(* PLC project mtcs_safety, Institute of Astronomy Onto 0.0.1 *)
(* stored: creationDateTime 2024-10-22T16:57:18.797943, modificationDateTime 2024-10-22T16:57:18.797943 *)

TYPE SafetyParts : STRUCT
  hydraulics : SafetyHydraulics;  (* Hydraulics safety *)
  emergencyStops : SafetyEmergencyStops;  (* Emergency stops *)
  domeAccess : SafetyDomeAccess;  (* Dome access *)
  motionBlocking : SafetyMotionBlocking;  (* Motion blocking *)
  domeShutter : SafetyDomeShutter;  (* Dome Shutter *)
  io : SafetyIO;  (* I/O modules *)
  configManager : ConfigManager;  (* The config manager (to load/save/activate configuration data) *)
END_STRUCT;
END_TYPE

TYPE SafetyIOParts : STRUCT
  domeAccess : SafetyDomeAccessIO;  (* DA: Dome access I/O *)
  hydraulicsAndSafety : SafetyHydraulicsAndSafetyIO;  (* HS: Hydraulics and Safety I/O *)
END_STRUCT;
END_TYPE

TYPE SafetyHydraulicsAndSafetyIOParts : STRUCT
  COU : EtherCatDevice;  (* HS:COU (EK1101) *)
  DO1 : EtherCatDevice;  (* HS:DO1 (EL2008) *)
  SI1 : EtherCatDevice;  (* HS:SI1 (EL1904) *)
  SI2 : EtherCatDevice;  (* HS:SI2 (EL1904) *)
  SI3 : EtherCatDevice;  (* HS:SI3 (EL1904) *)
  SI4 : EtherCatDevice;  (* HS:SI4 (EL1904) *)
  SL : EtherCatDevice;  (* HS:SL (EL6900) *)
  SO1 : EtherCatDevice;  (* HS:SO1 (EL2904) *)
  AI1 : EtherCatDevice;  (* HS:AI1 (EL3102) *)
  AI2 : EtherCatDevice;  (* HS:AI2 (EL3152) *)
  RTD1 : EtherCatDevice;  (* HS:RTD1 (EL3202-0010) *)
  PWR1 : EtherCatDevice;  (* HS:PWR1 (EL9410) *)
  AO1 : EtherCatDevice;  (* HS:AO1 (EL4132) *)
END_STRUCT;
END_TYPE

TYPE SafetyDomeAccessIOParts : STRUCT
  COU : EtherCatDevice;  (* DA:COU (EK1101) *)
  DI1 : EtherCatDevice;  (* DA:DI1 (EL1008) *)
  DI2 : EtherCatDevice;  (* DA:DI2 (EL1008) *)
  DO1 : EtherCatDevice;  (* DA:DO1 (EL2008) *)
  SI1 : EtherCatDevice;  (* DA:SI1 (EL1904) *)
  RE1 : EtherCatDevice;  (* DA:RE1 (EL2622) *)
  RE2 : EtherCatDevice;  (* DA:RE2 (EL2622) *)
END_STRUCT;
END_TYPE

TYPE SafetyDomeAccessParts : STRUCT
  lampsRelay1 : SimpleRelay;  (* Lamps relay 1 *)
  lampsRelay2 : SimpleRelay;  (* Lamps relay 2 *)
  lampsRelay3 : SimpleRelay;  (* Lamps relay 3 *)
  lampsRelay4 : SimpleRelay;  (* Lamps relay 4 *)
END_STRUCT;
END_TYPE

TYPE SafetyProcesses : STRUCT
  initialize : Process;  (* Start initializing *)
  lock : Process;  (* Lock the system *)
  unlock : Process;  (* Unlock the system *)
  changeOperatingState : ChangeOperatingStateProcess;  (* Change the operating state (e.g. AUTO, MANUAL, ...) *)
END_STRUCT;
END_TYPE

TYPE SafetyHydraulicsProcesses : STRUCT
  startupPumps : Process;  (* Start up the pumps (this will first trigger a reset() command!) *)
  reset : Process;  (* Reset the errors (including the programmed ones and the TwinSAFE group ones) *)
END_STRUCT;
END_TYPE

TYPE SafetyEmergencyStopsProcesses : STRUCT
  reset : Process;  (* Reset the errors (including the programmed ones and the TwinSAFE group ones) *)
END_STRUCT;
END_TYPE

TYPE SafetyDomeAccessProcesses : STRUCT
  reset : Process;  (* Reset the errors (including the programmed ones and the TwinSAFE group ones) *)
  personHasLeft : Process;  (* Unblock the telescope (if possible, i.e. if no E-Stops are active etc.) *)
  bypass : Process;  (* Bypass the doors sensors for the number of seconds defined in the config *)
  bypassPermanently : Process;  (* Bypass the doors sensors permanently (until re-initialization) *)
  stopBypassing : Process;  (* Stop bypassing the doors sensors *)
END_STRUCT;
END_TYPE

TYPE SafetyMotionBlockingProcesses : STRUCT
  reset : Process;  (* Reset the errors (including the programmed ones and the TwinSAFE group ones) *)
END_STRUCT;
END_TYPE

TYPE SafetyDomeShutterProcesses : STRUCT
  reset : Process;  (* Reset the errors (including the programmed ones and the TwinSAFE group ones) *)
END_STRUCT;
END_TYPE

TYPE SafetyStatuses : STRUCT
  initializationStatus : InitializationStatus;
  healthStatus : HealthStatus;
  busyStatus : BusyStatus;
  operatingStatus : OperatingStatus;
  communicationHealthStatus : HealthStatus;
  functionBlockHealthStatus : HealthStatus;
  outputHealthStatus : HealthStatus;
END_STRUCT;
END_TYPE

TYPE SafetyIOStatuses : STRUCT
  healthStatus : HealthStatus;  (* Is the I/O in a healthy state? *)
END_STRUCT;
END_TYPE

TYPE SafetyHydraulicsAndSafetyIOStatuses : STRUCT
  healthStatus : HealthStatus;  (* Is the I/O in a healthy state? *)
END_STRUCT;
END_TYPE

TYPE SafetyDomeAccessIOStatuses : STRUCT
  healthStatus : HealthStatus;  (* Is the I/O in a healthy state? *)
END_STRUCT;
END_TYPE

TYPE SafetyHydraulicsStatuses : STRUCT
  healthStatus : HealthStatus;  (* Is the safety in a healthy state? Good=RUN, Bad=safe stopped *)
  busyStatus : BusyStatus;  (* Is the safety busy? *)
END_STRUCT;
END_TYPE

TYPE SafetyEmergencyStopsStatuses : STRUCT
  healthStatus : HealthStatus;  (* Are the emergency stops in a healthy state? Good=RUN, Bad=safe stopped *)
  busyStatus : BusyStatus;  (* Is the safety busy? *)
END_STRUCT;
END_TYPE

TYPE SafetyDomeAccessStatuses : STRUCT
  healthStatus : HealthStatus;  (* Are the emergency stops in a healthy state? Good=RUN, Bad=safe stopped *)
  busyStatus : BusyStatus;  (* Is the safety busy? *)
END_STRUCT;
END_TYPE

TYPE SafetyMotionBlockingStatuses : STRUCT
  busyStatus : BusyStatus;  (* Is the safety busy? *)
  healthStatus : HealthStatus;  (* Is everything unblocked? Good=unblocked, Bad=safe stopped *)
END_STRUCT;
END_TYPE

TYPE SafetyDomeShutterStatuses : STRUCT
  busyStatus : BusyStatus;  (* Is the safety busy? *)
  healthStatus : HealthStatus;  (* Is everything unblocked? Good=unblocked, Bad=safe stopped *)
END_STRUCT;
END_TYPE

TYPE SafetyDomeAccessAlertConfig : STRUCT
  pattern : UDINT;  (* Bit pattern, for which bit=high means alert active, bit=low means alert off *)
  patternLength : USINT;  (* Number of bits of the bitPattern to use (between 1 and 32) *)
  bitLength : UINT;  (* Sound length of 1 bit, in milliseconds *)
  totalTime : UINT;  (* The time, in number of milliseconds, during which the pattern is repeated. 0 means repeat forever. *)
END_STRUCT;
END_TYPE

TYPE SafetyDomeAccessConfig : STRUCT
  disabled : BOOL;  (* True if the dome access control system should be disabled permanently. *)
  bypassTimeAfterPassword : LREAL;  (* Time until during which the doors sensors are being bypassed after entering the password, in seconds *)
  bypassingSound : SafetyDomeAccessAlertConfig;  (* Sound to play when the doors sensors are being bypassed *)
  bypassedPermanentlyVisual : SafetyDomeAccessAlertConfig;  (* LED pattern to play when the doors sensors are now bypassed permanently *)
  doorsOpenedWhenEnteringSound : SafetyDomeAccessAlertConfig;  (* Sound to play when a door is being opened for the first time (i.e. when a person is entering) *)
  doorsOpenedWhenLeavingSound : SafetyDomeAccessAlertConfig;  (* Sound to play when a door is being opened for the 2nd or 3rd or ... time (i.e. when a person is leaving) *)
  leavingWhenDoorsClosedSound : SafetyDomeAccessAlertConfig;  (* Sound to play when the personHasLeftButton is pressed when the doors are closed *)
  leavingWhenDoosOpenedSound : SafetyDomeAccessAlertConfig;  (* Sound to play when the personHasLeftButton is pressed when the doors are still open *)
  doorsOpenedVisual : SafetyDomeAccessAlertConfig;  (* LED pattern to play when the doors were opened without bypass (i.e. without password) *)
END_STRUCT;
END_TYPE

TYPE SafetyConfig : STRUCT
  domeAccess : SafetyDomeAccessConfig;  (* Some configuration values of the Dome Access *)
END_STRUCT;
END_TYPE

FUNCTION_BLOCK SM_Safety
  VAR_INPUT
    {attribute 'OPC.UA.DA' := '1'}
    {attribute 'OPC.UA.DA.Access' := '1'}
    editableConfig : SafetyConfig;  (* Editable configuration of the Safety subsystem *)
  END_VAR
  VAR_OUTPUT
    {attribute 'OPC.UA.DA' := '1'}
    {attribute 'OPC.UA.DA.Access' := '1'}
    actualStatus : STRING;  (* Current status description *)
    previousStatus : STRING;  (* Previous status description *)
    {attribute 'OPC.UA.DA' := '1'}
    {attribute 'OPC.UA.DA.Access' := '1'}
    config : SafetyConfig;  (* Active configuration of the Safety subsystem *)
    statuses : SafetyStatuses;  (* Statuses of the state machine *)
    parts : SafetyParts;  (* Parts of the state machine *)
    processes : SafetyProcesses;  (* Processes of the state machine *)
  END_VAR
  VAR_IN_OUT
    {attribute 'OPC.UA.DA' := '0'}
    operatorStatus : OperatorStatus;  (* Shared operator status *)
    {attribute 'OPC.UA.DA' := '0'}
    activityStatus : ActivityStatus;  (* Shared activity status *)
  END_VAR

            parts.hydraulics(
    operatorStatus := operatorStatus,
    activityStatus := activityStatus);
parts.emergencyStops();
parts.domeAccess(
    operatorStatus := operatorStatus,
    activityStatus := activityStatus,
    config := config.domeAccess);
parts.motionBlocking(
    activityStatus := activityStatus,
    hydraulics := parts.hydraulics,
    emergencyStops := parts.emergencyStops,
    domeAccess := parts.domeAccess);
parts.domeShutter(
    activityStatus := activityStatus,
    emergencyStops := parts.emergencyStops);
parts.io();
parts.configManager( isEnabled := operatorStatus.tech );
statuses.initializationStatus();
statuses.healthStatus(
    isGood := parts.io.statuses.healthStatus.isGood AND (parts.hydraulics.statuses.healthStatus.isGood AND (parts.emergencyStops.statuses.healthStatus.isGood AND (parts.domeAccess.statuses.healthStatus.isGood AND (parts.motionBlocking.statuses.healthStatus.isGood AND parts.domeShutter.statuses.healthStatus.isGood)))),
    hasWarning := parts.io.statuses.healthStatus.hasWarning OR (parts.hydraulics.statuses.healthStatus.hasWarning OR (parts.emergencyStops.statuses.healthStatus.hasWarning OR (parts.domeAccess.statuses.healthStatus.hasWarning OR (parts.motionBlocking.statuses.healthStatus.hasWarning OR parts.domeShutter.statuses.healthStatus.hasWarning)))));
statuses.busyStatus( isBusy := statuses.initializationStatus.initializing OR (parts.emergencyStops.statuses.busyStatus.busy OR (parts.domeAccess.statuses.busyStatus.busy OR (parts.hydraulics.statuses.busyStatus.busy OR (parts.domeShutter.statuses.busyStatus.busy OR parts.motionBlocking.statuses.busyStatus.busy)))) );
statuses.operatingStatus( superState := statuses.initializationStatus.initialized );
statuses.communicationHealthStatus();
statuses.functionBlockHealthStatus();
statuses.outputHealthStatus();
processes.initialize( isEnabled := statuses.initializationStatus.shutdown OR (statuses.initializationStatus.initializingFailed OR statuses.initializationStatus.initialized) );
processes.lock( isEnabled := operatorStatus.tech AND statuses.initializationStatus.initialized );
processes.unlock( isEnabled := operatorStatus.tech AND statuses.initializationStatus.locked );
processes.changeOperatingState( isEnabled := FALSE );

          

{attribute 'TcRpcEnable' := '1'}
METHOD initialize : RequestResults
                  initialize := THIS^.processes.initialize.request();

                
END_METHOD

{attribute 'TcRpcEnable' := '1'}
METHOD lock : RequestResults
                  lock := THIS^.processes.lock.request();

                
END_METHOD

{attribute 'TcRpcEnable' := '1'}
METHOD unlock : RequestResults
                  unlock := THIS^.processes.unlock.request();

                
END_METHOD

{attribute 'TcRpcEnable' := '1'}
METHOD changeOperatingState : RequestResults
  VAR_INPUT
    state : OperatingStates;
  END_VAR
                  changeOperatingState := THIS^.processes.changeOperatingState.request( state := state );

                
END_METHOD

{attribute 'TcRpcEnable' := '1'}
METHOD _log : BOOL
  VAR_INPUT
    name : STRING;  (* Name of this function block instance *)
  END_VAR
  VAR_IN_OUT
    buffer : LogBuffer;  (* Buffer to write all logging to *)
  END_VAR
  VAR
    subBuffer : LogBuffer;  (* Temporary buffer to write logging by parts (sub-statemachines) to *)
  END_VAR
                  THIS^.parts.hydraulics._log(
    name := 'hydraulics',
    buffer := subBuffer);
THIS^.parts.emergencyStops._log(
    name := 'emergencyStops',
    buffer := subBuffer);
THIS^.parts.domeAccess._log(
    name := 'domeAccess',
    buffer := subBuffer);
THIS^.parts.motionBlocking._log(
    name := 'motionBlocking',
    buffer := subBuffer);
THIS^.parts.domeShutter._log(
    name := 'domeShutter',
    buffer := subBuffer);
THIS^.parts.io._log(
    name := 'io',
    buffer := subBuffer);
THIS^.parts.configManager._log(
    name := 'configManager',
    buffer := subBuffer);
THIS^.processes.initialize._log(
    name := 'processes.initialize',
    buffer := subBuffer);
THIS^.processes.lock._log(
    name := 'processes.lock',
    buffer := subBuffer);
THIS^.processes.unlock._log(
    name := 'processes.unlock',
    buffer := subBuffer);
THIS^.processes.changeOperatingState._log(
    name := 'processes.changeOperatingState',
    buffer := subBuffer);
LOGGER(
    name := name,
    actualStatus := THIS^.actualStatus,
    previousStatus := THIS^.previousStatus,
    buffer := buffer,
    subBuffer := subBuffer,
    pHealthStatus := ADR(THIS^.statuses.healthStatus),
    pBusyStatus := ADR(THIS^.statuses.busyStatus));

                
END_METHOD
END_FUNCTION_BLOCK

FUNCTION_BLOCK SM_SafetyIO
  VAR_OUTPUT
    {attribute 'OPC.UA.DA' := '1'}
    {attribute 'OPC.UA.DA.Access' := '1'}
    actualStatus : STRING;  (* Current status description *)
    previousStatus : STRING;  (* Previous status description *)
    statuses : SafetyIOStatuses;  (* Statuses of the state machine *)
    parts : SafetyIOParts;  (* Parts of the state machine *)
  END_VAR

            parts.domeAccess();
parts.hydraulicsAndSafety();
statuses.healthStatus(
    isGood := parts.hydraulicsAndSafety.statuses.healthStatus.isGood AND parts.domeAccess.statuses.healthStatus.isGood,
    hasWarning := parts.hydraulicsAndSafety.statuses.healthStatus.hasWarning OR parts.domeAccess.statuses.healthStatus.hasWarning);

          

{attribute 'TcRpcEnable' := '1'}
METHOD _log : BOOL
  VAR_INPUT
    name : STRING;  (* Name of this function block instance *)
  END_VAR
  VAR_IN_OUT
    buffer : LogBuffer;  (* Buffer to write all logging to *)
  END_VAR
  VAR
    subBuffer : LogBuffer;  (* Temporary buffer to write logging by parts (sub-statemachines) to *)
  END_VAR
                  THIS^.parts.domeAccess._log(
    name := 'domeAccess',
    buffer := subBuffer);
THIS^.parts.hydraulicsAndSafety._log(
    name := 'hydraulicsAndSafety',
    buffer := subBuffer);
LOGGER(
    name := name,
    actualStatus := THIS^.actualStatus,
    previousStatus := THIS^.previousStatus,
    buffer := buffer,
    subBuffer := subBuffer,
    pHealthStatus := ADR(THIS^.statuses.healthStatus));

                
END_METHOD
END_FUNCTION_BLOCK

FUNCTION_BLOCK SM_SafetyHydraulicsAndSafetyIO
  VAR_OUTPUT
    {attribute 'OPC.UA.DA' := '1'}
    {attribute 'OPC.UA.DA.Access' := '1'}
    actualStatus : STRING;  (* Current status description *)
    previousStatus : STRING;  (* Previous status description *)
    statuses : SafetyHydraulicsAndSafetyIOStatuses;  (* Statuses of the state machine *)
    parts : SafetyHydraulicsAndSafetyIOParts;  (* Parts of the state machine *)
  END_VAR

            parts.COU(
    id := 'HS:COU',
    typeId := 'EK1101');
parts.DO1(
    id := 'HS:DI1',
    typeId := 'EL2008');
parts.SI1(
    id := 'HS:SI1',
    typeId := 'EL1904');
parts.SI2(
    id := 'HS:SI2',
    typeId := 'EL1904');
parts.SI3(
    id := 'HS:SI3',
    typeId := 'EL1904');
parts.SI4(
    id := 'HS:SI3',
    typeId := 'EL1904');
parts.SL(
    id := 'HS:SL',
    typeId := 'EL6900');
parts.SO1(
    id := 'HS:SO1',
    typeId := 'EL2904');
parts.AI1(
    id := 'HS:AI1',
    typeId := 'EL3102');
parts.AI2(
    id := 'HS:AI2',
    typeId := 'EL3152');
parts.RTD1(
    id := 'HS:RTD1',
    typeId := 'EL3202-0010');
parts.PWR1(
    id := 'HS:PWR1',
    typeId := 'EL9410');
parts.AO1(
    id := 'HS:AO1',
    typeId := 'EL4132');
statuses.healthStatus(
    isGood := parts.COU.statuses.healthStatus.isGood AND (parts.DO1.statuses.healthStatus.isGood AND (parts.SI1.statuses.healthStatus.isGood AND (parts.SI2.statuses.healthStatus.isGood AND (parts.SI3.statuses.healthStatus.isGood AND (parts.SI4.statuses.healthStatus.isGood AND (parts.SL.statuses.healthStatus.isGood AND (parts.SO1.statuses.healthStatus.isGood AND (parts.AI1.statuses.healthStatus.isGood AND (parts.AI2.statuses.healthStatus.isGood AND (parts.RTD1.statuses.healthStatus.isGood AND (parts.PWR1.statuses.healthStatus.isGood AND parts.AO1.statuses.healthStatus.isGood))))))))))),
    hasWarning := parts.COU.statuses.healthStatus.hasWarning OR (parts.DO1.statuses.healthStatus.hasWarning OR (parts.SI1.statuses.healthStatus.hasWarning OR (parts.SI2.statuses.healthStatus.hasWarning OR (parts.SI3.statuses.healthStatus.hasWarning OR (parts.SI4.statuses.healthStatus.hasWarning OR (parts.SL.statuses.healthStatus.hasWarning OR (parts.SO1.statuses.healthStatus.hasWarning OR (parts.AI1.statuses.healthStatus.hasWarning OR (parts.AI2.statuses.healthStatus.hasWarning OR (parts.RTD1.statuses.healthStatus.hasWarning OR (parts.PWR1.statuses.healthStatus.hasWarning OR parts.AO1.statuses.healthStatus.hasWarning))))))))))));

          

{attribute 'TcRpcEnable' := '1'}
METHOD _log : BOOL
  VAR_INPUT
    name : STRING;  (* Name of this function block instance *)
  END_VAR
  VAR_IN_OUT
    buffer : LogBuffer;  (* Buffer to write all logging to *)
  END_VAR
  VAR
    subBuffer : LogBuffer;  (* Temporary buffer to write logging by parts (sub-statemachines) to *)
  END_VAR
                  THIS^.parts.COU._log(
    name := 'COU',
    buffer := subBuffer);
THIS^.parts.DO1._log(
    name := 'DO1',
    buffer := subBuffer);
THIS^.parts.SI1._log(
    name := 'SI1',
    buffer := subBuffer);
THIS^.parts.SI2._log(
    name := 'SI2',
    buffer := subBuffer);
THIS^.parts.SI3._log(
    name := 'SI3',
    buffer := subBuffer);
THIS^.parts.SI4._log(
    name := 'SI4',
    buffer := subBuffer);
THIS^.parts.SL._log(
    name := 'SL',
    buffer := subBuffer);
THIS^.parts.SO1._log(
    name := 'SO1',
    buffer := subBuffer);
THIS^.parts.AI1._log(
    name := 'AI1',
    buffer := subBuffer);
THIS^.parts.AI2._log(
    name := 'AI2',
    buffer := subBuffer);
THIS^.parts.RTD1._log(
    name := 'RTD1',
    buffer := subBuffer);
THIS^.parts.PWR1._log(
    name := 'PWR1',
    buffer := subBuffer);
THIS^.parts.AO1._log(
    name := 'AO1',
    buffer := subBuffer);
LOGGER(
    name := name,
    actualStatus := THIS^.actualStatus,
    previousStatus := THIS^.previousStatus,
    buffer := buffer,
    subBuffer := subBuffer,
    pHealthStatus := ADR(THIS^.statuses.healthStatus));

                
END_METHOD
END_FUNCTION_BLOCK

FUNCTION_BLOCK SM_SafetyDomeAccessIO
  VAR_OUTPUT
    {attribute 'OPC.UA.DA' := '1'}
    {attribute 'OPC.UA.DA.Access' := '1'}
    actualStatus : STRING;  (* Current status description *)
    previousStatus : STRING;  (* Previous status description *)
    statuses : SafetyDomeAccessIOStatuses;  (* Statuses of the state machine *)
    parts : SafetyDomeAccessIOParts;  (* Parts of the state machine *)
  END_VAR

            parts.COU(
    id := 'DA:COU',
    typeId := 'EK1101');
parts.DI1(
    id := 'DA:DI1',
    typeId := 'EL1008');
parts.DI2(
    id := 'DA:DI2',
    typeId := 'EL1008');
parts.DO1(
    id := 'DA:DO1',
    typeId := 'EL2008');
parts.SI1(
    id := 'DA:SI1',
    typeId := 'EL1904');
parts.RE1(
    id := 'DA:RE1',
    typeId := 'EL2622');
parts.RE2(
    id := 'DA:RE2',
    typeId := 'EL2622');
statuses.healthStatus(
    isGood := parts.COU.statuses.healthStatus.isGood AND (parts.DI1.statuses.healthStatus.isGood AND (parts.DI2.statuses.healthStatus.isGood AND (parts.DO1.statuses.healthStatus.isGood AND (parts.SI1.statuses.healthStatus.isGood AND (parts.RE1.statuses.healthStatus.isGood AND parts.RE2.statuses.healthStatus.isGood))))),
    hasWarning := parts.COU.statuses.healthStatus.hasWarning OR (parts.DI1.statuses.healthStatus.hasWarning OR (parts.DI2.statuses.healthStatus.hasWarning OR (parts.DO1.statuses.healthStatus.hasWarning OR (parts.SI1.statuses.healthStatus.hasWarning OR (parts.RE1.statuses.healthStatus.hasWarning OR parts.RE2.statuses.healthStatus.hasWarning))))));

          

{attribute 'TcRpcEnable' := '1'}
METHOD _log : BOOL
  VAR_INPUT
    name : STRING;  (* Name of this function block instance *)
  END_VAR
  VAR_IN_OUT
    buffer : LogBuffer;  (* Buffer to write all logging to *)
  END_VAR
  VAR
    subBuffer : LogBuffer;  (* Temporary buffer to write logging by parts (sub-statemachines) to *)
  END_VAR
                  THIS^.parts.COU._log(
    name := 'COU',
    buffer := subBuffer);
THIS^.parts.DI1._log(
    name := 'DI1',
    buffer := subBuffer);
THIS^.parts.DI2._log(
    name := 'DI2',
    buffer := subBuffer);
THIS^.parts.DO1._log(
    name := 'DO1',
    buffer := subBuffer);
THIS^.parts.SI1._log(
    name := 'SI1',
    buffer := subBuffer);
THIS^.parts.RE1._log(
    name := 'RE1',
    buffer := subBuffer);
THIS^.parts.RE2._log(
    name := 'RE2',
    buffer := subBuffer);
LOGGER(
    name := name,
    actualStatus := THIS^.actualStatus,
    previousStatus := THIS^.previousStatus,
    buffer := buffer,
    subBuffer := subBuffer,
    pHealthStatus := ADR(THIS^.statuses.healthStatus));

                
END_METHOD
END_FUNCTION_BLOCK

FUNCTION_BLOCK SM_SafetyHydraulics
  VAR_INPUT
    {attribute 'OPC.UA.DA' := '1'}
    {attribute 'OPC.UA.DA.Access' := '1'}
    groupComError AT %I* : BOOL;  (* TwinSAFE group communication error *)
    {attribute 'OPC.UA.DA' := '1'}
    {attribute 'OPC.UA.DA.Access' := '1'}
    groupFbError AT %I* : BOOL;  (* TwinSAFE group function block error *)
    {attribute 'OPC.UA.DA' := '1'}
    {attribute 'OPC.UA.DA.Access' := '1'}
    groupOutError AT %I* : BOOL;  (* TwinSAFE group output error *)
    {attribute 'OPC.UA.DA' := '1'}
    {attribute 'OPC.UA.DA.Access' := '1'}
    pumpsPowered AT %I* : BOOL;  (* TRUE if the pumps are powered *)
    {attribute 'OPC.UA.DA' := '1'}
    {attribute 'OPC.UA.DA.Access' := '1'}
    returnFilterOverpressure AT %I* : BOOL;  (* TRUE if the oil return filter has an overpressure *)
    {attribute 'OPC.UA.DA' := '1'}
    {attribute 'OPC.UA.DA.Access' := '1'}
    pumpsMinFrequency AT %I* : BOOL;  (* TRUE if the pumps run at a minimum frequency (frequency > QMin) *)
    {attribute 'OPC.UA.DA' := '1'}
    {attribute 'OPC.UA.DA.Access' := '1'}
    pumpsFrequencyNotRising AT %I* : BOOL;  (* TRUE if the frequency of the pumps is not rising after a startup command *)
    {attribute 'OPC.UA.DA' := '1'}
    {attribute 'OPC.UA.DA.Access' := '1'}
    pressureNotRising AT %I* : BOOL;  (* TRUE if the pressure is not rising after the frequency is rising *)
    {attribute 'OPC.UA.DA' := '1'}
    {attribute 'OPC.UA.DA.Access' := '1'}
    top1NoUnderpressure AT %I* : BOOL;  (* TRUE if there is no underpressure for Top pipe 1 *)
    {attribute 'OPC.UA.DA' := '1'}
    {attribute 'OPC.UA.DA.Access' := '1'}
    top2NoUnderpressure AT %I* : BOOL;  (* TRUE if there is no underpressure for Top pipe 2 *)
    {attribute 'OPC.UA.DA' := '1'}
    {attribute 'OPC.UA.DA.Access' := '1'}
    top3NoUnderpressure AT %I* : BOOL;  (* TRUE if there is no underpressure for Top pipe 3 *)
    {attribute 'OPC.UA.DA' := '1'}
    {attribute 'OPC.UA.DA.Access' := '1'}
    top4NoUnderpressure AT %I* : BOOL;  (* TRUE if there is no underpressure for Top pipe 4 *)
    {attribute 'OPC.UA.DA' := '1'}
    {attribute 'OPC.UA.DA.Access' := '1'}
    bottom5NoUnderpressure AT %I* : BOOL;  (* TRUE if there is no underpressure for Bottom pipe 5 *)
    {attribute 'OPC.UA.DA' := '1'}
    {attribute 'OPC.UA.DA.Access' := '1'}
    bottom6NoUnderpressure AT %I* : BOOL;  (* TRUE if there is no underpressure for Bottom pipe 6 *)
    {attribute 'OPC.UA.DA' := '1'}
    {attribute 'OPC.UA.DA.Access' := '1'}
    bottom7NoUnderpressure AT %I* : BOOL;  (* TRUE if there is no underpressure for Bottom pipe 7 *)
    {attribute 'OPC.UA.DA' := '1'}
    {attribute 'OPC.UA.DA.Access' := '1'}
    bottom8NoUnderpressure AT %I* : BOOL;  (* TRUE if there is no underpressure for Bottom pipe 8 *)
    {attribute 'OPC.UA.DA' := '1'}
    {attribute 'OPC.UA.DA.Access' := '1'}
    topNoOverpressure AT %I* : BOOL;  (* TRUE if there is no overpressure for the Top pipes *)
    {attribute 'OPC.UA.DA' := '1'}
    {attribute 'OPC.UA.DA.Access' := '1'}
    bottomNoOverpressure AT %I* : BOOL;  (* TRUE if there is no overpressure for the Bottom pipes *)
    {attribute 'OPC.UA.DA' := '1'}
    {attribute 'OPC.UA.DA.Access' := '1'}
    topTripOK AT %I* : BOOL;  (* TRUE if there is no TRIP error for the top drive *)
    {attribute 'OPC.UA.DA' := '1'}
    {attribute 'OPC.UA.DA.Access' := '1'}
    bottomTripOK AT %I* : BOOL;  (* TRUE if there is no overpressure for the botton drive *)
    {attribute 'OPC.UA.DA' := '1'}
    {attribute 'OPC.UA.DA.Access' := '1'}
    noUnderpressure AT %I* : BOOL;  (* TRUE if there is no underpressure for all 8 pipes *)
    {attribute 'OPC.UA.DA' := '1'}
    {attribute 'OPC.UA.DA.Access' := '1'}
    noUnderpressureNoDelay AT %I* : BOOL;  (* TRUE if there is no underpressure for all 8 pipes (even momentarily, without delay) *)
    {attribute 'OPC.UA.DA' := '1'}
    {attribute 'OPC.UA.DA.Access' := '1'}
    underpressureError AT %I* : BOOL;  (* TRUE if there is an underpressure problem (e.g. when the pumps are running and there is an underpressure) *)
    {attribute 'OPC.UA.DA' := '1'}
    {attribute 'OPC.UA.DA.Access' := '1'}
    noOverpressure AT %I* : BOOL;  (* TRUE if there is no overpressure for all 8 pipes *)
    {attribute 'OPC.UA.DA' := '1'}
    {attribute 'OPC.UA.DA.Access' := '1'}
    pumpsStartingUp AT %I* : BOOL;  (* TRUE if the pumps are restarting *)
    {attribute 'OPC.UA.DA' := '1'}
    {attribute 'OPC.UA.DA.Access' := '1'}
    pumpsStopped AT %I* : BOOL;  (* TRUE if the pumps are stopped *)
    {attribute 'OPC.UA.DA' := '1'}
    {attribute 'OPC.UA.DA.Access' := '1'}
    pumpsRunning AT %I* : BOOL;  (* TRUE if the pumps are running *)
    {attribute 'OPC.UA.DA' := '1'}
    {attribute 'OPC.UA.DA.Access' := '1'}
    pumpsRelease AT %I* : BOOL;  (* TRUE if the pumps are released (RFR 'ReglerFreigabe' high) *)
    {attribute 'OPC.UA.DA' := '1'}
    {attribute 'OPC.UA.DA.Access' := '1'}
    allOK AT %I* : BOOL;  (* TRUE if the hydraulics are OK *)
  END_VAR
  VAR_OUTPUT
    {attribute 'OPC.UA.DA' := '1'}
    {attribute 'OPC.UA.DA.Access' := '1'}
    actualStatus : STRING;  (* Current status description *)
    previousStatus : STRING;  (* Previous status description *)
    {attribute 'OPC.UA.DA' := '1'}
    {attribute 'OPC.UA.DA.Access' := '1'}
    restartPumpsOutput AT %Q* : BOOL;  (* Output to restart the pumps *)
    {attribute 'OPC.UA.DA' := '1'}
    {attribute 'OPC.UA.DA.Access' := '1'}
    resetErrorsOutput AT %Q* : BOOL;  (* Output to reset the errors *)
    {attribute 'OPC.UA.DA' := '1'}
    {attribute 'OPC.UA.DA.Access' := '1'}
    errorAcknowledge AT %Q* : BOOL;  (* Output to restart the TwinSAFE group *)
    statuses : SafetyHydraulicsStatuses;  (* Statuses of the state machine *)
    processes : SafetyHydraulicsProcesses;  (* Processes of the state machine *)
  END_VAR
  VAR_IN_OUT
    {attribute 'OPC.UA.DA' := '0'}
    operatorStatus : OperatorStatus;  (* Shared operator status *)
    {attribute 'OPC.UA.DA' := '0'}
    activityStatus : ActivityStatus;  (* Shared activity status *)
  END_VAR

            statuses.healthStatus( isGood := allOK AND (NOT(groupComError OR (groupFbError OR groupOutError))) );
statuses.busyStatus( isBusy := processes.startupPumps.statuses.busyStatus.busy OR processes.reset.statuses.busyStatus.busy );
processes.startupPumps( isEnabled := (NOT(pumpsStartingUp OR processes.startupPumps.statuses.busyStatus.busy)) AND operatorStatus.tech );
processes.reset( isEnabled := NOT(processes.reset.statuses.busyStatus.busy) );

          

{attribute 'TcRpcEnable' := '1'}
METHOD startupPumps : RequestResults
                  startupPumps := THIS^.processes.startupPumps.request();

                
END_METHOD

{attribute 'TcRpcEnable' := '1'}
METHOD reset : RequestResults
                  reset := THIS^.processes.reset.request();

                
END_METHOD

{attribute 'TcRpcEnable' := '1'}
METHOD _log : BOOL
  VAR_INPUT
    name : STRING;  (* Name of this function block instance *)
  END_VAR
  VAR_IN_OUT
    buffer : LogBuffer;  (* Buffer to write all logging to *)
  END_VAR
  VAR
    subBuffer : LogBuffer;  (* Temporary buffer to write logging by parts (sub-statemachines) to *)
  END_VAR
                  THIS^.processes.startupPumps._log(
    name := 'processes.startupPumps',
    buffer := subBuffer);
THIS^.processes.reset._log(
    name := 'processes.reset',
    buffer := subBuffer);
LOGGER(
    name := name,
    actualStatus := THIS^.actualStatus,
    previousStatus := THIS^.previousStatus,
    buffer := buffer,
    subBuffer := subBuffer,
    pHealthStatus := ADR(THIS^.statuses.healthStatus),
    pBusyStatus := ADR(THIS^.statuses.busyStatus));

                
END_METHOD
END_FUNCTION_BLOCK

FUNCTION_BLOCK SM_SafetyEmergencyStops
  VAR_INPUT
    {attribute 'OPC.UA.DA' := '1'}
    {attribute 'OPC.UA.DA.Access' := '1'}
    groupComError AT %I* : BOOL;  (* TwinSAFE group communication error *)
    {attribute 'OPC.UA.DA' := '1'}
    {attribute 'OPC.UA.DA.Access' := '1'}
    groupFbError AT %I* : BOOL;  (* TwinSAFE group function block error *)
    {attribute 'OPC.UA.DA' := '1'}
    {attribute 'OPC.UA.DA.Access' := '1'}
    groupOutError AT %I* : BOOL;  (* TwinSAFE group output error *)
    {attribute 'OPC.UA.DA' := '1'}
    {attribute 'OPC.UA.DA.Access' := '1'}
    allOK AT %I* : BOOL;  (* TRUE if the emergency stops are OK *)
    {attribute 'OPC.UA.DA' := '1'}
    {attribute 'OPC.UA.DA.Access' := '1'}
    discrepancyError AT %I* : BOOL;  (* TRUE if there is a discrepancy time error between two contacts of an emergency stop *)
    {attribute 'OPC.UA.DA' := '1'}
    {attribute 'OPC.UA.DA.Access' := '1'}
    dome1NO AT %I* : BOOL;  (* TRUE if the make contact (NO) is conducting --> button is pushed! *)
    {attribute 'OPC.UA.DA' := '1'}
    {attribute 'OPC.UA.DA.Access' := '1'}
    dome1NC AT %I* : BOOL;  (* TRUE if the break contact (NC) is conducting --> button is not pushed *)
    {attribute 'OPC.UA.DA' := '1'}
    {attribute 'OPC.UA.DA.Access' := '1'}
    dome2NO AT %I* : BOOL;  (* TRUE if the make contact (NO) is conducting --> button is pushed! *)
    {attribute 'OPC.UA.DA' := '1'}
    {attribute 'OPC.UA.DA.Access' := '1'}
    dome2NC AT %I* : BOOL;  (* TRUE if the break contact (NC) is conducting --> button is not pushed *)
    {attribute 'OPC.UA.DA' := '1'}
    {attribute 'OPC.UA.DA.Access' := '1'}
    firstFloorNO AT %I* : BOOL;  (* TRUE if the make contact (NO) is conducting --> button is pushed! *)
    {attribute 'OPC.UA.DA' := '1'}
    {attribute 'OPC.UA.DA.Access' := '1'}
    firstFloorNC AT %I* : BOOL;  (* TRUE if the break contact (NC) is conducting --> button is not pushed *)
    {attribute 'OPC.UA.DA' := '1'}
    {attribute 'OPC.UA.DA.Access' := '1'}
    controlRoomNO AT %I* : BOOL;  (* TRUE if the make contact (NO) is conducting --> button is pushed! *)
    {attribute 'OPC.UA.DA' := '1'}
    {attribute 'OPC.UA.DA.Access' := '1'}
    controlRoomNC AT %I* : BOOL;  (* TRUE if the break contact (NC) is conducting --> button is not pushed *)
    {attribute 'OPC.UA.DA' := '1'}
    {attribute 'OPC.UA.DA.Access' := '1'}
    domeAccessNO AT %I* : BOOL;  (* TRUE if the make contact (NO) is conducting --> button is pushed! *)
    {attribute 'OPC.UA.DA' := '1'}
    {attribute 'OPC.UA.DA.Access' := '1'}
    domeAccessNC AT %I* : BOOL;  (* TRUE if the break contact (NC) is conducting --> button is not pushed *)
  END_VAR
  VAR_OUTPUT
    {attribute 'OPC.UA.DA' := '1'}
    {attribute 'OPC.UA.DA.Access' := '1'}
    actualStatus : STRING;  (* Current status description *)
    previousStatus : STRING;  (* Previous status description *)
    {attribute 'OPC.UA.DA' := '1'}
    {attribute 'OPC.UA.DA.Access' := '1'}
    restartOutput AT %Q* : BOOL;  (* Output to restart the emergency buttons *)
    {attribute 'OPC.UA.DA' := '1'}
    {attribute 'OPC.UA.DA.Access' := '1'}
    errorAcknowledge AT %Q* : BOOL;  (* Output to restart the TwinSAFE group *)
    statuses : SafetyEmergencyStopsStatuses;  (* Statuses of the state machine *)
    processes : SafetyEmergencyStopsProcesses;  (* Processes of the state machine *)
  END_VAR

            statuses.healthStatus( isGood := allOK AND (NOT(groupComError OR (groupFbError OR (groupOutError OR discrepancyError)))) );
statuses.busyStatus( isBusy := processes.reset.statuses.busyStatus.busy );
processes.reset( isEnabled := NOT(processes.reset.statuses.busyStatus.busy) );

          

{attribute 'TcRpcEnable' := '1'}
METHOD reset : RequestResults
                  reset := THIS^.processes.reset.request();

                
END_METHOD

{attribute 'TcRpcEnable' := '1'}
METHOD _log : BOOL
  VAR_INPUT
    name : STRING;  (* Name of this function block instance *)
  END_VAR
  VAR_IN_OUT
    buffer : LogBuffer;  (* Buffer to write all logging to *)
  END_VAR
  VAR
    subBuffer : LogBuffer;  (* Temporary buffer to write logging by parts (sub-statemachines) to *)
  END_VAR
                  THIS^.processes.reset._log(
    name := 'processes.reset',
    buffer := subBuffer);
LOGGER(
    name := name,
    actualStatus := THIS^.actualStatus,
    previousStatus := THIS^.previousStatus,
    buffer := buffer,
    subBuffer := subBuffer,
    pHealthStatus := ADR(THIS^.statuses.healthStatus),
    pBusyStatus := ADR(THIS^.statuses.busyStatus));

                
END_METHOD
END_FUNCTION_BLOCK

FUNCTION_BLOCK SM_SafetyDomeAccess
  VAR_INPUT
    {attribute 'OPC.UA.DA' := '1'}
    {attribute 'OPC.UA.DA.Access' := '1'}
    groupComError AT %I* : BOOL;  (* TwinSAFE group communication error *)
    {attribute 'OPC.UA.DA' := '1'}
    {attribute 'OPC.UA.DA.Access' := '1'}
    groupFbError AT %I* : BOOL;  (* TwinSAFE group function block error *)
    {attribute 'OPC.UA.DA' := '1'}
    {attribute 'OPC.UA.DA.Access' := '1'}
    groupOutError AT %I* : BOOL;  (* TwinSAFE group output error *)
    {attribute 'OPC.UA.DA' := '1'}
    {attribute 'OPC.UA.DA.Access' := '1'}
    keypadKey1 AT %I* : BOOL;  (* TRUE if keypad key 1 is being pressed *)
    {attribute 'OPC.UA.DA' := '1'}
    {attribute 'OPC.UA.DA.Access' := '1'}
    keypadKey2 AT %I* : BOOL;  (* TRUE if keypad key 2 is being pressed *)
    {attribute 'OPC.UA.DA' := '1'}
    {attribute 'OPC.UA.DA.Access' := '1'}
    keypadKey3 AT %I* : BOOL;  (* TRUE if keypad key 3 is being pressed *)
    {attribute 'OPC.UA.DA' := '1'}
    {attribute 'OPC.UA.DA.Access' := '1'}
    keypadKey4 AT %I* : BOOL;  (* TRUE if keypad key 4 is being pressed *)
    {attribute 'OPC.UA.DA' := '1'}
    {attribute 'OPC.UA.DA.Access' := '1'}
    keypadKey5 AT %I* : BOOL;  (* TRUE if keypad key 5 is being pressed *)
    {attribute 'OPC.UA.DA' := '1'}
    {attribute 'OPC.UA.DA.Access' := '1'}
    keypadKey6 AT %I* : BOOL;  (* TRUE if keypad key 6 is being pressed *)
    {attribute 'OPC.UA.DA' := '1'}
    {attribute 'OPC.UA.DA.Access' := '1'}
    keypadKey7 AT %I* : BOOL;  (* TRUE if keypad key 7 is being pressed *)
    {attribute 'OPC.UA.DA' := '1'}
    {attribute 'OPC.UA.DA.Access' := '1'}
    keypadKey8 AT %I* : BOOL;  (* TRUE if keypad key 8 is being pressed *)
    {attribute 'OPC.UA.DA' := '1'}
    {attribute 'OPC.UA.DA.Access' := '1'}
    keypadKey9 AT %I* : BOOL;  (* TRUE if keypad key 9 is being pressed *)
    {attribute 'OPC.UA.DA' := '1'}
    {attribute 'OPC.UA.DA.Access' := '1'}
    keypadKeyStar AT %I* : BOOL;  (* TRUE if keypad key * is being pressed *)
    {attribute 'OPC.UA.DA' := '1'}
    {attribute 'OPC.UA.DA.Access' := '1'}
    door1Closed AT %I* : BOOL;  (* TRUE if door 1 is closed *)
    {attribute 'OPC.UA.DA' := '1'}
    {attribute 'OPC.UA.DA.Access' := '1'}
    door2Closed AT %I* : BOOL;  (* TRUE if door 2 is closed *)
    {attribute 'OPC.UA.DA' := '1'}
    {attribute 'OPC.UA.DA.Access' := '1'}
    personHasLeftButtonPressed AT %I* : BOOL;  (* TRUE if the unblock button is being pressed *)
    {attribute 'OPC.UA.DA' := '1'}
    {attribute 'OPC.UA.DA.Access' := '1'}
    returnButtonPressed AT %I* : BOOL;  (* TRUE if the return button is being pressed *)
    {attribute 'OPC.UA.DA' := '1'}
    {attribute 'OPC.UA.DA.Access' := '1'}
    safeAccess AT %I* : BOOL;  (* TRUE if the safety still allows motion (e.g. also during the first seconds that a person has entered *)
  END_VAR
  VAR_OUTPUT
    {attribute 'OPC.UA.DA' := '1'}
    {attribute 'OPC.UA.DA.Access' := '1'}
    actualStatus : STRING;  (* Current status description *)
    previousStatus : STRING;  (* Previous status description *)
    {attribute 'OPC.UA.DA' := '1'}
    {attribute 'OPC.UA.DA.Access' := '1'}
    errorAcknowledge AT %Q* : BOOL;  (* Output to restart the TwinSAFE group *)
    {attribute 'OPC.UA.DA' := '1'}
    {attribute 'OPC.UA.DA.Access' := '1'}
    personHasEntered AT %Q* : BOOL;  (* TRUE if the doors were opened without bypass/password *)
    {attribute 'OPC.UA.DA' := '1'}
    {attribute 'OPC.UA.DA.Access' := '1'}
    enteredLedOn AT %Q* : BOOL;  (* TRUE if the yellow led should be on *)
    {attribute 'OPC.UA.DA' := '1'}
    {attribute 'OPC.UA.DA.Access' := '1'}
    movingLedOn AT %Q* : BOOL;  (* TRUE if the red led should be on *)
    {attribute 'OPC.UA.DA' := '1'}
    {attribute 'OPC.UA.DA.Access' := '1'}
    awakeLedOn AT %Q* : BOOL;  (* TRUE if the yellow led should be on *)
    {attribute 'OPC.UA.DA' := '1'}
    {attribute 'OPC.UA.DA.Access' := '1'}
    sleepingLedOn AT %Q* : BOOL;  (* TRUE if the orange led should be on *)
    {attribute 'OPC.UA.DA' := '1'}
    {attribute 'OPC.UA.DA.Access' := '1'}
    buzzerSounding AT %Q* : BOOL;  (* TRUE if the green is being sounded *)
    {attribute 'OPC.UA.DA' := '1'}
    {attribute 'OPC.UA.DA.Access' := '1'}
    sensorsBeingBypassed : BOOL;  (* TRUE if the sensors are currently being bypassed *)
    {attribute 'OPC.UA.DA' := '1'}
    {attribute 'OPC.UA.DA.Access' := '1'}
    sensorsBypassedPermanently : BOOL;  (* TRUE if the sensors are being bypassed permanently *)
    statuses : SafetyDomeAccessStatuses;  (* Statuses of the state machine *)
    parts : SafetyDomeAccessParts;  (* Parts of the state machine *)
    processes : SafetyDomeAccessProcesses;  (* Processes of the state machine *)
  END_VAR
  VAR_IN_OUT
    {attribute 'OPC.UA.DA' := '0'}
    operatorStatus : OperatorStatus;  (* Shared operator status *)
    {attribute 'OPC.UA.DA' := '0'}
    activityStatus : ActivityStatus;  (* Shared activity status *)
    {attribute 'OPC.UA.DA' := '0'}
    config : SafetyDomeAccessConfig;  (* The dome access config *)
  END_VAR

            parts.lampsRelay1( isEnabled := operatorStatus.tech );
parts.lampsRelay2( isEnabled := operatorStatus.tech );
parts.lampsRelay3( isEnabled := operatorStatus.tech );
parts.lampsRelay4( isEnabled := operatorStatus.tech );
statuses.healthStatus(
    isGood := NOT(groupComError OR (groupFbError OR groupOutError)),
    hasWarning := personHasEntered OR sensorsBypassedPermanently);
statuses.busyStatus( isBusy := processes.reset.statuses.busyStatus.busy OR (processes.personHasLeft.statuses.busyStatus.busy OR (processes.bypass.statuses.busyStatus.busy OR (processes.bypassPermanently.statuses.busyStatus.busy OR processes.stopBypassing.statuses.busyStatus.busy))) );
processes.reset( isEnabled := statuses.busyStatus.idle );
processes.personHasLeft( isEnabled := statuses.busyStatus.idle AND operatorStatus.tech );
processes.bypass( isEnabled := statuses.busyStatus.idle AND (operatorStatus.tech AND (NOT(sensorsBeingBypassed))) );
processes.bypassPermanently( isEnabled := statuses.busyStatus.idle AND (operatorStatus.tech AND (NOT(sensorsBypassedPermanently))) );
processes.stopBypassing( isEnabled := statuses.busyStatus.idle AND (operatorStatus.tech AND (sensorsBeingBypassed OR sensorsBypassedPermanently)) );

          

{attribute 'TcRpcEnable' := '1'}
METHOD reset : RequestResults
                  reset := THIS^.processes.reset.request();

                
END_METHOD

{attribute 'TcRpcEnable' := '1'}
METHOD personHasLeft : RequestResults
                  personHasLeft := THIS^.processes.personHasLeft.request();

                
END_METHOD

{attribute 'TcRpcEnable' := '1'}
METHOD bypass : RequestResults
                  bypass := THIS^.processes.bypass.request();

                
END_METHOD

{attribute 'TcRpcEnable' := '1'}
METHOD bypassPermanently : RequestResults
                  bypassPermanently := THIS^.processes.bypassPermanently.request();

                
END_METHOD

{attribute 'TcRpcEnable' := '1'}
METHOD stopBypassing : RequestResults
                  stopBypassing := THIS^.processes.stopBypassing.request();

                
END_METHOD

{attribute 'TcRpcEnable' := '1'}
METHOD _log : BOOL
  VAR_INPUT
    name : STRING;  (* Name of this function block instance *)
  END_VAR
  VAR_IN_OUT
    buffer : LogBuffer;  (* Buffer to write all logging to *)
  END_VAR
  VAR
    subBuffer : LogBuffer;  (* Temporary buffer to write logging by parts (sub-statemachines) to *)
  END_VAR
                  THIS^.parts.lampsRelay1._log(
    name := 'lampsRelay1',
    buffer := subBuffer);
THIS^.parts.lampsRelay2._log(
    name := 'lampsRelay2',
    buffer := subBuffer);
THIS^.parts.lampsRelay3._log(
    name := 'lampsRelay3',
    buffer := subBuffer);
THIS^.parts.lampsRelay4._log(
    name := 'lampsRelay4',
    buffer := subBuffer);
THIS^.processes.reset._log(
    name := 'processes.reset',
    buffer := subBuffer);
THIS^.processes.personHasLeft._log(
    name := 'processes.personHasLeft',
    buffer := subBuffer);
THIS^.processes.bypass._log(
    name := 'processes.bypass',
    buffer := subBuffer);
THIS^.processes.bypassPermanently._log(
    name := 'processes.bypassPermanently',
    buffer := subBuffer);
THIS^.processes.stopBypassing._log(
    name := 'processes.stopBypassing',
    buffer := subBuffer);
LOGGER(
    name := name,
    actualStatus := THIS^.actualStatus,
    previousStatus := THIS^.previousStatus,
    buffer := buffer,
    subBuffer := subBuffer,
    pHealthStatus := ADR(THIS^.statuses.healthStatus),
    pBusyStatus := ADR(THIS^.statuses.busyStatus));

                
END_METHOD
END_FUNCTION_BLOCK

FUNCTION_BLOCK SM_SafetyMotionBlocking
  VAR_INPUT
    {attribute 'OPC.UA.DA' := '1'}
    {attribute 'OPC.UA.DA.Access' := '1'}
    groupComError AT %I* : BOOL;  (* TwinSAFE group communication error *)
    {attribute 'OPC.UA.DA' := '1'}
    {attribute 'OPC.UA.DA.Access' := '1'}
    groupFbError AT %I* : BOOL;  (* TwinSAFE group function block error *)
    {attribute 'OPC.UA.DA' := '1'}
    {attribute 'OPC.UA.DA.Access' := '1'}
    groupOutError AT %I* : BOOL;  (* TwinSAFE group output error *)
    {attribute 'OPC.UA.DA' := '1'}
    {attribute 'OPC.UA.DA.Access' := '1'}
    telescopeAzimuthReleaseOK AT %I* : BOOL;  (* TRUE if the telescope azimuth axis is released *)
    {attribute 'OPC.UA.DA' := '1'}
    {attribute 'OPC.UA.DA.Access' := '1'}
    telescopeElevationReleaseOK AT %I* : BOOL;  (* TRUE if the telescope elevation axis is released *)
    {attribute 'OPC.UA.DA' := '1'}
    {attribute 'OPC.UA.DA.Access' := '1'}
    telescopeRotationReleaseOK AT %I* : BOOL;  (* TRUE if the telescope rotation axes are released *)
    {attribute 'OPC.UA.DA' := '1'}
    {attribute 'OPC.UA.DA.Access' := '1'}
    domeRotationReleaseOK AT %I* : BOOL;  (* TRUE if the dome rotation axis is released *)
    {attribute 'OPC.UA.DA' := '1'}
    {attribute 'OPC.UA.DA.Access' := '1'}
    motionAllowed AT %I* : BOOL;  (* TRUE if motion is allowed *)
  END_VAR
  VAR_OUTPUT
    {attribute 'OPC.UA.DA' := '1'}
    {attribute 'OPC.UA.DA.Access' := '1'}
    actualStatus : STRING;  (* Current status description *)
    previousStatus : STRING;  (* Previous status description *)
    {attribute 'OPC.UA.DA' := '1'}
    {attribute 'OPC.UA.DA.Access' := '1'}
    errorAcknowledge AT %Q* : BOOL;  (* Output to restart the TwinSAFE group *)
    statuses : SafetyMotionBlockingStatuses;  (* Statuses of the state machine *)
    processes : SafetyMotionBlockingProcesses;  (* Processes of the state machine *)
  END_VAR
  VAR_IN_OUT
    {attribute 'OPC.UA.DA' := '0'}
    activityStatus : ActivityStatus;  (* Shared activity status *)
    {attribute 'OPC.UA.DA' := '0'}
    hydraulics : SafetyHydraulics;
    {attribute 'OPC.UA.DA' := '0'}
    emergencyStops : SafetyEmergencyStops;
    {attribute 'OPC.UA.DA' := '0'}
    domeAccess : SafetyDomeAccess;
  END_VAR

            statuses.busyStatus( isBusy := processes.reset.statuses.busyStatus.busy );
statuses.healthStatus(
    isGood := NOT(groupComError OR (groupFbError OR groupOutError)),
    hasWarning := (activityStatus.awake OR activityStatus.moving) AND (NOT(telescopeAzimuthReleaseOK AND (telescopeElevationReleaseOK AND (telescopeRotationReleaseOK AND domeRotationReleaseOK)))));
processes.reset( isEnabled := NOT(processes.reset.statuses.busyStatus.busy) );

          

{attribute 'TcRpcEnable' := '1'}
METHOD reset : RequestResults
                  reset := THIS^.processes.reset.request();

                
END_METHOD

{attribute 'TcRpcEnable' := '1'}
METHOD _log : BOOL
  VAR_INPUT
    name : STRING;  (* Name of this function block instance *)
  END_VAR
  VAR_IN_OUT
    buffer : LogBuffer;  (* Buffer to write all logging to *)
  END_VAR
  VAR
    subBuffer : LogBuffer;  (* Temporary buffer to write logging by parts (sub-statemachines) to *)
  END_VAR
                  THIS^.processes.reset._log(
    name := 'processes.reset',
    buffer := subBuffer);
LOGGER(
    name := name,
    actualStatus := THIS^.actualStatus,
    previousStatus := THIS^.previousStatus,
    buffer := buffer,
    subBuffer := subBuffer,
    pHealthStatus := ADR(THIS^.statuses.healthStatus),
    pBusyStatus := ADR(THIS^.statuses.busyStatus));

                
END_METHOD
END_FUNCTION_BLOCK

FUNCTION_BLOCK SM_SafetyDomeShutter
  VAR_INPUT
    {attribute 'OPC.UA.DA' := '1'}
    {attribute 'OPC.UA.DA.Access' := '1'}
    groupComError AT %I* : BOOL;  (* TwinSAFE group communication error *)
    {attribute 'OPC.UA.DA' := '1'}
    {attribute 'OPC.UA.DA.Access' := '1'}
    groupFbError AT %I* : BOOL;  (* TwinSAFE group function block error *)
    {attribute 'OPC.UA.DA' := '1'}
    {attribute 'OPC.UA.DA.Access' := '1'}
    groupOutError AT %I* : BOOL;  (* TwinSAFE group output error *)
    {attribute 'OPC.UA.DA' := '1'}
    {attribute 'OPC.UA.DA.Access' := '1'}
    shutterAllowed AT %I* : BOOL;  (* TRUE if dome shutter is allowed *)
    {attribute 'OPC.UA.DA' := '1'}
    {attribute 'OPC.UA.DA.Access' := '1'}
    lowerOpenSafeOutput AT %I* : BOOL;  (* Safety open lower shutter command *)
    {attribute 'OPC.UA.DA' := '1'}
    {attribute 'OPC.UA.DA.Access' := '1'}
    lowerCloseSafeOutput AT %I* : BOOL;  (* Safety close lower shutter command *)
    {attribute 'OPC.UA.DA' := '1'}
    {attribute 'OPC.UA.DA.Access' := '1'}
    upperOpenSafeOutput AT %I* : BOOL;  (* Safety open upper shutter command *)
    {attribute 'OPC.UA.DA' := '1'}
    {attribute 'OPC.UA.DA.Access' := '1'}
    upperCloseSafeOutput AT %I* : BOOL;  (* Safety close upper shutter command *)
    {attribute 'OPC.UA.DA' := '1'}
    {attribute 'OPC.UA.DA.Access' := '1'}
    pumpOnSafeOutput AT %I* : BOOL;  (* Safety pump on command *)
  END_VAR
  VAR_OUTPUT
    {attribute 'OPC.UA.DA' := '1'}
    {attribute 'OPC.UA.DA.Access' := '1'}
    actualStatus : STRING;  (* Current status description *)
    previousStatus : STRING;  (* Previous status description *)
    {attribute 'OPC.UA.DA' := '1'}
    {attribute 'OPC.UA.DA.Access' := '1'}
    errorAcknowledge AT %Q* : BOOL;  (* Output to restart the TwinSAFE group *)
    statuses : SafetyDomeShutterStatuses;  (* Statuses of the state machine *)
    processes : SafetyDomeShutterProcesses;  (* Processes of the state machine *)
  END_VAR
  VAR_IN_OUT
    {attribute 'OPC.UA.DA' := '0'}
    activityStatus : ActivityStatus;  (* Shared activity status *)
    {attribute 'OPC.UA.DA' := '0'}
    emergencyStops : SafetyEmergencyStops;
  END_VAR

            statuses.busyStatus( isBusy := processes.reset.statuses.busyStatus.busy );
statuses.healthStatus( isGood := NOT(groupComError OR (groupFbError OR groupOutError)) );
processes.reset( isEnabled := NOT(processes.reset.statuses.busyStatus.busy) );

          

{attribute 'TcRpcEnable' := '1'}
METHOD reset : RequestResults
                  reset := THIS^.processes.reset.request();

                
END_METHOD

{attribute 'TcRpcEnable' := '1'}
METHOD _log : BOOL
  VAR_INPUT
    name : STRING;  (* Name of this function block instance *)
  END_VAR
  VAR_IN_OUT
    buffer : LogBuffer;  (* Buffer to write all logging to *)
  END_VAR
  VAR
    subBuffer : LogBuffer;  (* Temporary buffer to write logging by parts (sub-statemachines) to *)
  END_VAR
                  THIS^.processes.reset._log(
    name := 'processes.reset',
    buffer := subBuffer);
LOGGER(
    name := name,
    actualStatus := THIS^.actualStatus,
    previousStatus := THIS^.previousStatus,
    buffer := buffer,
    subBuffer := subBuffer,
    pHealthStatus := ADR(THIS^.statuses.healthStatus),
    pBusyStatus := ADR(THIS^.statuses.busyStatus));

                
END_METHOD
END_FUNCTION_BLOCK
